Fanuc KAREL source: kt00269.KL

PROGRAM KT00269
%STACKSIZE=65535
%PRIORITY=65535
%NOLOCKGROUP
VAR
OUT : BOOLEAN
-- UNRESOLVED DECLARATIONS (source type spelling not recovered)
-- Y1 : ARRAY[2] OF TYPE_0x0018 (type_u16=0x2018)
-- Y2 : ARRAY[2] OF TYPE_0x0018 (type_u16=0x2018)
BEGIN
Y1[1]=2
Y2[1]=3
Y1[1]=2
Y2[1]=3
-- UNRESOLVED_PC line 12 opcodes [22 9D 33 B1 22 9D 33 B1 57 23] marker_code=76
END KT00269
